// TwinCAT 3 PLC project LED_test
// ProgramVersion: 3.1.4022.7
// libraries:
//   Tc2_Standard, * (Beckhoff Automation GmbH)
//   Tc2_System, * (Beckhoff Automation GmbH)
//   Tc3_Module, * (Beckhoff Automation GmbH)
//   LCLS General,2.4.2,SLAC
// project tree:
//   / PlcTask.TcTTO
//   POUs/Function Blocks/ FB_AnalogOut.TcPOU, FB_PWM_Output.TcPOU, FB_TMO_LED.TcPOU
//   POUs/ MAIN.TcPOU
// real-time tasks:
//   TASK PlcTask: cycle T#10ms, priority 20, ADS port 350
// I/O:
//   DEVICE Device 1 (EtherCAT), AmsNetId 172.21.148.67.2.1
//     Power_EK1200 [EK1200-5000 EtherCAT Power supply (2A E-Bus)]
//       PWM_EL2502 [EL2502 2Ch. PWM output, 24V]
//       AO_EL4004 [EL4004 4Ch. Ana. Output 0-10V, 12bit]
//       Term 4 (EL9011) [EL9011 End Terminal]
// variable links:
//   LED_test/LED_test Instance <-> Device 1 (EtherCAT)/Power_EK1200/AO_EL4004
//     PlcTask Outputs/MAIN.bAnalogOutPut4.iRaw <-> AO Outputs Channel 4/Analog output
//     PlcTask Outputs/MAIN.bAnalogOutput1.iRaw <-> AO Outputs Channel 1/Analog output
//     PlcTask Outputs/MAIN.bAnalogOutput2.iRaw <-> AO Outputs Channel 2/Analog output
//     PlcTask Outputs/MAIN.bAnalogOutput3.iRaw <-> AO Outputs Channel 3/Analog output
//   LED_test/LED_test Instance <-> Device 1 (EtherCAT)/Power_EK1200/PWM_EL2502
//     PlcTask Outputs/MAIN.bPwmOutput1.iIlluminatorINT <-> PWM Outputs Channel 1/PWM output
//     PlcTask Outputs/MAIN.bPwmOutput2.iIlluminatorINT <-> PWM Outputs Channel 2/PWM output

CONFIGURATION LED_test
    RESOURCE PLC ON TwinCAT3
        TASK PlcTask(INTERVAL := T#10ms, PRIORITY := 20);
        PROGRAM MAIN WITH PlcTask : MAIN;
    END_RESOURCE
END_CONFIGURATION

// ---- POUs/MAIN.TcPOU
PROGRAM MAIN
VAR
	
// Analog Output variables

	{attribute 'TcLinkTo' := '.iRaw := TIID^Device 1 (EtherCAT)^Power_EK1200^AO_EL4004^AO Outputs Channel 1^Analog output'}
	bAnalogOutput1 : FB_AnalogOutput;
	
	{attribute 'TcLinkTo' := '.iRaw := TIID^Device 1 (EtherCAT)^Power_EK1200^AO_EL4004^AO Outputs Channel 2^Analog output'}
	bAnalogOutput2 : FB_AnalogOutput;
	
	{attribute 'TcLinkTo' := '.iRaw := TIID^Device 1 (EtherCAT)^Power_EK1200^AO_EL4004^AO Outputs Channel 3^Analog output'}
	bAnalogOutput3 : FB_AnalogOutput;
	
	{attribute 'TcLinkTo' := '.iRaw := TIID^Device 1 (EtherCAT)^Power_EK1200^AO_EL4004^AO Outputs Channel 4^Analog output'}
    bAnalogOutPut4 : FB_AnalogOutput;

	
// PWM Output variables
    {attribute 'TcLinkTo' := '.iIlluminatorINT := TIID^Device 1 (EtherCAT)^Power_EK1200^PWM_EL2502^PWM Outputs Channel 1^PWM output'}
    {attribute 'pytmc' := '
		pv: TST:01
		io: io
	'}
    bPwmOutput1 : FB_TMO_LED;	
	
	{attribute 'TcLinkTo' := '.iIlluminatorINT := TIID^Device 1 (EtherCAT)^Power_EK1200^PWM_EL2502^PWM Outputs Channel 2^PWM output'}
	{attribute 'pytmc' := '
		pv: TST:02
		io: io
	'}
	bPwmOutput2 : FB_TMO_LED;	

END_VAR

//bPwmOutput1.fIlluminatorPercent:=not IO.bMyInput1;

bPwmOutput1.M_Set_IllPercentage(100);
bPwmOutput1(fbSetIllPercent=>);

END_PROGRAM

// ---- POUs/Function Blocks/FB_TMO_LED.TcPOU
FUNCTION_BLOCK FB_TMO_LED
VAR
	iIlluminatorINT AT %Q*: INT;

    {attribute 'pytmc' := '
        pv: PWR
        field: ZNAM OFF
        field: ONAM ON
    '}
    bLedPower AT %Q*: BOOL;

    {attribute 'pytmc' := '
        pv: CIL:PCT
        EGU: %
    '}
    fIlluminatorPercent: LREAL;
//    fbGetIllPercent: FB_AnalogInput;
    fbSetIllPercent: FB_PWM_Output;

    bLedInit: BOOL := FALSE;
END_VAR

// Turn the LED off by default
IF bLedInit THEN
    bLedPower := FALSE;
//    bLedInit := TRUE;
END_IF

// Illuminator conversion to percentage
fbSetIllPercent(
    fReal:=fIlluminatorPercent,
    fSafeMax:=100,
    fSafeMin:=0,
    iTermBits:=14,
    fTermMax:=100,
    fTermMin:=0,
    iRaw=>iIlluminatorINT);

(*	
fbGetIllPercent(
    iRaw:=iIlluminatorINT,
    iTermBits:=15,
    fTermMax:=100,
    fTermMin:=0,
    fReal=>fIlluminatorPercent);
*)

METHOD M_Set_IllPercentage : LREAL
VAR_INPUT
	IlluminatorPercent : LREAL;
END_VAR
This^.fIlluminatorPercent := IlluminatorPercent;
END_METHOD

END_FUNCTION_BLOCK

// ---- POUs/Function Blocks/FB_PWM_Output.TcPOU
FUNCTION_BLOCK FB_PWM_Output
(*
	Converts a real unit value (e.g., volts) to the integer needed for a PWM output terminal.
	2022-04-26 Maarten Thomas-Bosum
*)

// The following was copied from FB_AnalogOutput so the variables need to be updated according
// to the specifications of the EL2502 PWM Output terminal.

VAR_INPUT
	// The real value to send to the output
	fReal: LREAL;
	// The maximum allowed real value for the connected hardware
	fSafeMax: LREAL;
	// The minimum allowed real value for the connected hardware
	fSafeMin: LREAL;
	// The number of bits correlated with the terminal's max output. This is not necessarily the resolution parameter.
	iTermBits: UINT;
	// The fReal value correlated with the terminal's max output
	fTermMax: LREAL;
	// The fReal value correlated with the terminal's min output
	fTermMin: LREAL;
END_VAR
VAR_OUTPUT
	// Connect this output to the terminal
	iRaw AT %Q*: INT;
END_VAR
VAR
	fScale: LREAL;
END_VAR

// Set the scaling from real to raw
IF fScale = 0 AND fTermMax > fTermMin THEN
	fScale := (EXPT(2, iTermBits) - 1) / (fTermMax - fTermMin);
END_IF

// Adjust real value to be within the limits
fReal := MIN(fReal, fSafeMax, fTermMax);
fReal := MAX(fReal, fSafeMin, fTermMin);

// Scale the output accordingly
iRaw := LREAL_TO_INT((fReal - fTermMin) * fScale);

END_FUNCTION_BLOCK

// ---- POUs/Function Blocks/FB_AnalogOut.TcPOU
FUNCTION_BLOCK FB_AnalogOut EXTENDS FB_AnalogOutput
VAR_INPUT
END_VAR
VAR_OUTPUT
END_VAR
VAR
END_VAR

END_FUNCTION_BLOCK
